// TIA Portal V17 export
// export: Created 2023-04-03T06:31:37.0714184Z, ExportSetting WithDefaults, DisplayName Totally Integrated Automation Portal, DisplayVersion V17 Update 4, DisplayName TIA Portal Openness, DisplayVersion V17 Update 4, DisplayName TIA Portal Version Control Interface, DisplayVersion V17, DisplayName STEP 7 Professional, DisplayVersion V17 Update 4, DisplayName STEP 7 Safety, DisplayVersion V17, DisplayName WinCC Professional, DisplayVersion V17 Update 4
ORGANIZATION_BLOCK "Cyclic interrupt 1s"   // OB35, LAD, CyclicInterrupt
{ S7_Optimized_Access := 'TRUE' }
VERSION : 0.1
// stored: AutoNumber false, IsIECCheckEnabled false, SetENOAutomatically false
   VAR_INPUT
      Initial_Call : Bool;   // Initial call of this OB
      Event_Count : Int;   // Events discarded
   END_VAR
BEGIN

REGION Network 1: Heartbeat BMS1
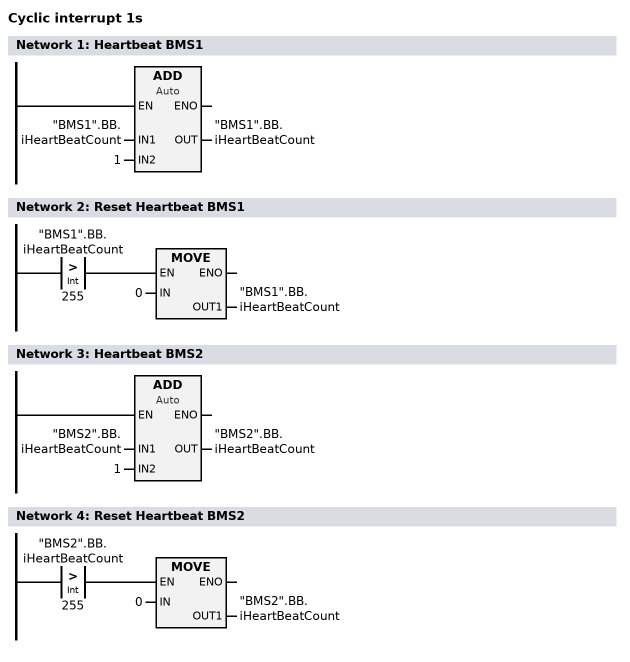
   RUNG wire#powerrail
      Add(in1 := "BMS1".BB.iHeartBeatCount, in2 := 1, out => "BMS1".BB.iHeartBeatCount)
   END_RUNG
   // the same network as SCL:
   "BMS1".BB.iHeartBeatCount := "BMS1".BB.iHeartBeatCount + 1;
END_REGION

REGION Network 2: Reset Heartbeat BMS1
   RUNG wire#powerrail
      { S7_Templates := "SrcType := Int" } GT_Contact(in1 := "BMS1".BB.iHeartBeatCount, in2 := 255)
      Move(in := 0, out1 => "BMS1".BB.iHeartBeatCount)
   END_RUNG
   // the same network as SCL:
   IF "BMS1".BB.iHeartBeatCount > 255 THEN "BMS1".BB.iHeartBeatCount := 0; END_IF;
END_REGION

REGION Network 3: Heartbeat BMS2
   RUNG wire#powerrail
      Add(in1 := "BMS2".BB.iHeartBeatCount, in2 := 1, out => "BMS2".BB.iHeartBeatCount)
   END_RUNG
   // the same network as SCL:
   "BMS2".BB.iHeartBeatCount := "BMS2".BB.iHeartBeatCount + 1;
END_REGION

REGION Network 4: Reset Heartbeat BMS2
   RUNG wire#powerrail
      { S7_Templates := "SrcType := Int" } GT_Contact(in1 := "BMS2".BB.iHeartBeatCount, in2 := 255)
      Move(in := 0, out1 => "BMS2".BB.iHeartBeatCount)
   END_RUNG
   // the same network as SCL:
   IF "BMS2".BB.iHeartBeatCount > 255 THEN "BMS2".BB.iHeartBeatCount := 0; END_IF;
END_REGION
END_ORGANIZATION_BLOCK
